FUNCTION_BLOCK svVerifyBoolLogic (* Basic Function Block Type *)
  (* Standard: 61499-2 *)
  (* Version 0.0, 3/4/2015, Bernd Glatz, nxtControl GmbH, Template *)
  PACKAGE Loytec.Automation;
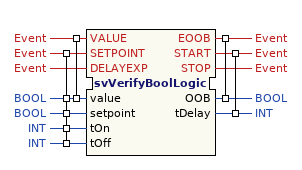
  EVENT_INPUT
    VALUE WITH value; (* Value input has changed *)
    SETPOINT WITH value, setpoint, tOn, tOff; (* Setpoint has changed *)
    DELAYEXP; (* Delay Expired *)
  END_EVENT
  EVENT_OUTPUT
    EOOB WITH OOB; (* OOB Event *)
    START WITH tDelay; (* Start delay event *)
    STOP; (* Stop delay event *)
  END_EVENT
  VAR_INPUT
    value : BOOL; (* Input value *)
    setpoint : BOOL; (* Setpoint *)
    tOn : INT; (* Granted time after setpoint becomes TRUE *)
    tOff : INT; (* Granted time after setpoint becomes FALSE *)
  END_VAR
  VAR_OUTPUT
    OOB : BOOL; (* Out of Bounds indication *)
    tDelay : INT; (* Time value for delay *)
  END_VAR
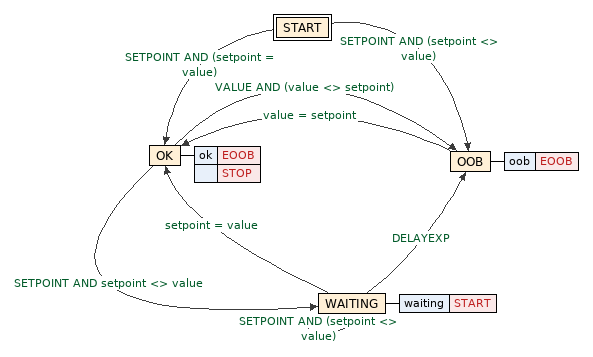
  EC_STATES
    START; (* Initial State *)
    OK : ok -> EOOB, -> STOP;
    WAITING : waiting -> START;
    OOB : oob -> EOOB;
  END_STATES
  EC_TRANSITIONS
    START TO OK := SETPOINT AND (setpoint = value);
    WAITING TO OOB := DELAYEXP;
    OK TO OOB := VALUE AND (value <> setpoint);
    OOB TO OK := value = setpoint;
    START TO OOB := SETPOINT AND (setpoint <> value);
    OK TO WAITING := SETPOINT AND setpoint <> value;
    WAITING TO OK := setpoint = value;
    WAITING TO WAITING := SETPOINT AND (setpoint <> value);
  END_TRANSITIONS
  ALGORITHM ok IN ST:
IF OOB THEN
	OOB := FALSE;
ELSE
	EOOB := FALSE;
END_IF;

IF tDelay <> 0 THEN
	tDelay := 0;
ELSE
	STOP := FALSE;
END_IF;
  END_ALGORITHM
  ALGORITHM waiting IN ST:
tDelay := SEL(setpoint, tOff, tOn);
SETPOINT := FALSE;
  END_ALGORITHM
  ALGORITHM oob IN ST:
IF NOT OOB THEN
	OOB := TRUE;
ELSE
	EOOB := FALSE;
END_IF;

IF tDelay <> 0 THEN
	tDelay := 0;
END_IF;
  END_ALGORITHM
END_FUNCTION_BLOCK
